Staubli VAL3: SetToolParam.pgx

program SetToolParam(num value)
  local num prevType
  local tool prevTool
  local bool inLimits
begin
  //*******************************************************************************
  //*   ______
  //*  / _____) /|
  //* | |      / /
  //* | | /\  / /
  //* | | \ \/ /  _      Copyright (c) KEOLABS, 2016
  //* | |  \__/  | |        http://www.keolabs.com
  //* | |________| |
  //*  \__________/
  //*
  //********************************************************************************
  //*@file          : SetToolParam
  //*@author        : Yves Ragot
  //*@version       : $Id: SetToolParam.pgx 1490 2016-12-14 15:39:12Z yves $
  //*@brief         : Set the length of the tool
  //*
  //*******************************************************************************/

  // save previous tool parameter
  prevTool = tCurrentTool
  prevType = currentToolType

  // set new tool
  tCurrentTool = flange
  tCurrentTool.trsf.z = value
  tCurrentTool.trsf.rx = -180
  tCurrentTool.trsf.rz = 180
  currentToolType = 99

  // check if current position with new tool is in new limits
  call IsInLimits(inLimits)

  // if not, error
  if (!inLimits)

      // restore previous limits
      tCurrentTool = prevTool
      currentToolType = prevType

      // parameter error
      GeneralStatus = 101
      LastErrorCode = 0

  endIf

end
